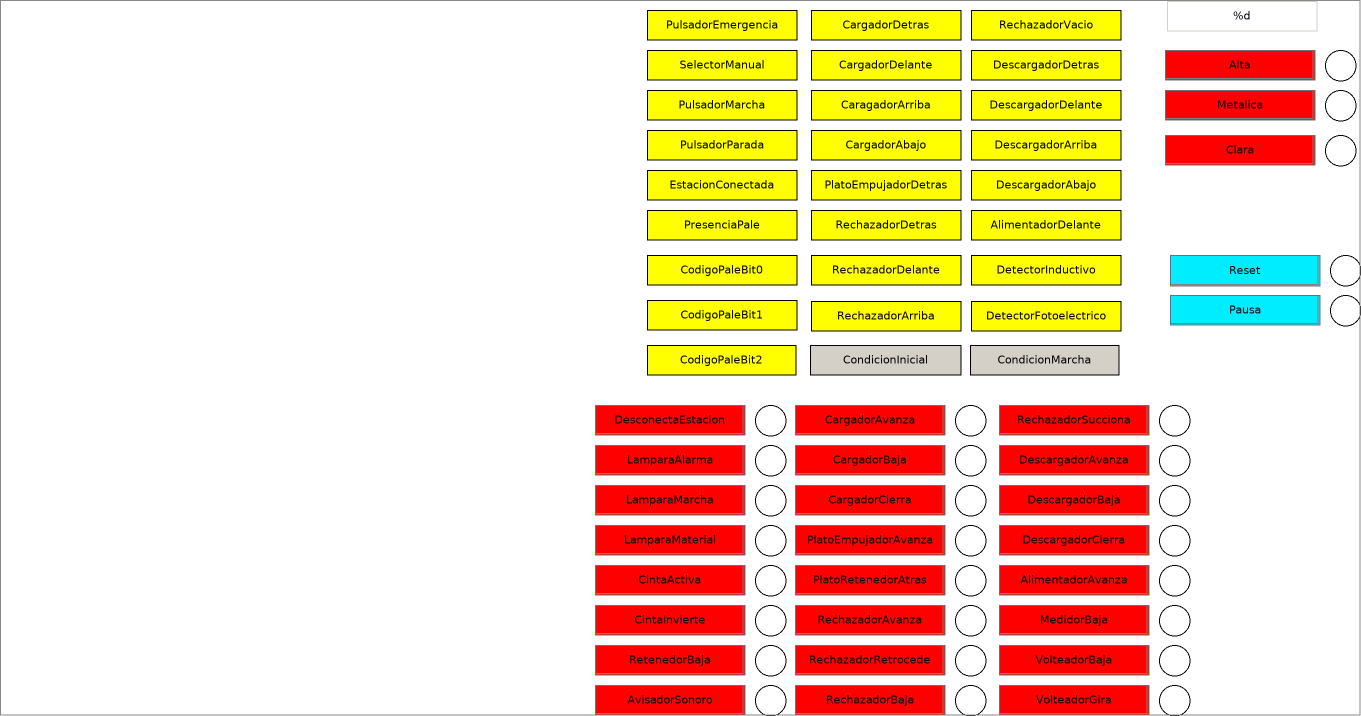
VISUALIZATION Visualization  // 1361x716
    Rectangle (647,170 150x30), "EstacionConectada", colour toggle: MAIN.Estacion.EstacionConectada
        toggle MAIN.Estacion.EstacionConectada
    Rectangle (647,210 150x30), "PresenciaPale", colour toggle: MAIN.Estacion.PresenciaPale
        toggle MAIN.Estacion.PresenciaPale
    Rectangle (647,255 150x30), "CodigoPaleBit0", colour toggle: MAIN.Estacion.CodigoPaleBit0
        toggle MAIN.Estacion.CodigoPaleBit0
    Rectangle (647,300 150x30), "CodigoPaleBit1", colour toggle: MAIN.Estacion.CodigoPaleBit1
        toggle MAIN.Estacion.CodigoPaleBit1
    Rectangle (647,345 149x30), "CodigoPaleBit2", colour toggle: MAIN.Estacion.CodigoPaleBit2
        toggle MAIN.Estacion.CodigoPaleBit2
    Rectangle (647,130 150x30), "PulsadorParada", colour toggle: MAIN.Estacion.PulsadorParada
        toggle MAIN.Estacion.PulsadorParada
    Rectangle (647,90 150x30), "PulsadorMarcha", colour toggle: MAIN.Estacion.PulsadorMarcha
        toggle MAIN.Estacion.PulsadorMarcha
    Rectangle (647,50 150x30), "SelectorManual", colour toggle: MAIN.Estacion.SelectorManual
        toggle MAIN.Estacion.SelectorManual
    Rectangle (647,10 150x30), "PulsadorEmergencia", colour toggle: MAIN.Estacion.PulsadorEmergencia
        toggle MAIN.Estacion.PulsadorEmergencia
    Rectangle (811,170 150x30), "PlatoEmpujadorDetras", colour toggle: MAIN.Estacion.PlatoEmpujadorDetras
        toggle MAIN.Estacion.PlatoEmpujadorDetras
    Rectangle (811,210 150x30), "RechazadorDetras", colour toggle: MAIN.Estacion.RechazadorDetras
        toggle MAIN.Estacion.RechazadorDetras
    Rectangle (811,255 150x30), "RechazadorDelante", colour toggle: MAIN.Estacion.RechazadorDelante
        toggle MAIN.Estacion.RechazadorDelante
    Rectangle (811,130 150x30), "CargadorAbajo", colour toggle: MAIN.Estacion.CargadorAbajo
        toggle MAIN.Estacion.CargadorAbajo
    Rectangle (811,90 150x30), "CaragadorArriba", colour toggle: MAIN.Estacion.CargadorArriba
        toggle MAIN.Estacion.CargadorArriba
    Rectangle (811,50 150x30), "CargadorDelante", colour toggle: MAIN.Estacion.CargadorDelante
        toggle MAIN.Estacion.CargadorDelante
    Rectangle (811,10 150x30), "CargadorDetras", colour toggle: MAIN.Estacion.CargadorDetras
        toggle MAIN.Estacion.CargadorDetras
    Rectangle (811,301 150x30), "RechazadorArriba", colour toggle: MAIN.Estacion.RechazadorArriba
        toggle MAIN.Estacion.RechazadorArriba
    Rectangle (971,170 150x30), "DescargadorAbajo", colour toggle: MAIN.Estacion.DescargadorAbajo
        toggle MAIN.Estacion.DescargadorAbajo
    Rectangle (971,210 150x30), "AlimentadorDelante", colour toggle: MAIN.Estacion.AlimentadorDelante
        toggle MAIN.Estacion.AlimentadorDelante
    Rectangle (971,255 150x30), "DetectorInductivo", colour toggle: MAIN.Estacion.DetectorInductivo
        toggle MAIN.Estacion.DetectorInductivo
    Rectangle (971,130 150x30), "DescargadorArriba", colour toggle: MAIN.Estacion.DescargadorArriba
        toggle MAIN.Estacion.DescargadorArriba
    Rectangle (971,90 150x30), "DescargadorDelante", colour toggle: MAIN.Estacion.DescargadorDelante
        toggle MAIN.Estacion.DescargadorDelante
    Rectangle (971,50 150x30), "DescargadorDetras", colour toggle: MAIN.Estacion.DescargadorDetras
        toggle MAIN.Estacion.DescargadorDetras
    Rectangle (971,10 150x30), "RechazadorVacio", colour toggle: MAIN.Estacion.RechazadorVacio
        toggle MAIN.Estacion.RechazadorVacio
    Rectangle (971,301 150x30), "DetectorFotoelectrico", colour toggle: MAIN.Estacion.DetectorFotoelectrico
        toggle MAIN.Estacion.DetectorFotoelectrico
    Rectangle (810,345 151x30), "CondicionInicial", colour toggle: MAIN.Estacion.CondicionInicial
        toggle MAIN.Estacion.CondicionInicial
    Rectangle (970,345 149x30), "CondicionMarcha", colour toggle: MAIN.Estacion.CondicionMarcha
        toggle MAIN.Estacion.CondicionMarcha
    Button (595,445 150x30), "LamparaAlarma"
        toggle MAIN.Estacion.LamparaAlarma
    Ellipse (755,445 31x31), colour toggle: MAIN.Estacion.LamparaAlarma
    Button (595,405 150x30), "DesconectaEstacion"
        toggle MAIN.Estacion.DesconectaEstacion
    Ellipse (755,405 31x31), colour toggle: MAIN.Estacion.DesconectaEstacion
    Button (595,525 150x30), "LamparaMaterial"
        toggle MAIN.Estacion.LamparaMaterial
    Ellipse (755,525 31x31), colour toggle: MAIN.Estacion.LamparaMaterial
    Button (595,485 150x30), "LamparaMarcha"
        toggle MAIN.Estacion.LamparaMarcha
    Ellipse (755,485 31x31), colour toggle: MAIN.Estacion.LamparaMarcha
    Button (595,605 150x30), "CintaInvierte"
        toggle MAIN.Estacion.CintaInvierte
    Ellipse (755,605 31x31), colour toggle: MAIN.Estacion.CintaInvierte
    Button (595,565 150x30), "CintaActiva"
        toggle MAIN.Estacion.CintaActiva
    Ellipse (755,565 31x31), colour toggle: MAIN.Estacion.CintaActiva
    Button (595,685 150x30), "AvisadorSonoro"
        toggle MAIN.Estacion.AvisadorSonoro
    Ellipse (755,685 31x31), colour toggle: MAIN.Estacion.AvisadorSonoro
    Button (595,645 150x30), "RetenedorBaja"
        toggle MAIN.Estacion.RetenedorBaja
    Ellipse (755,645 31x31), colour toggle: MAIN.Estacion.RetenedorBaja
    Button (795,445 150x30), "CargadorBaja"
        toggle MAIN.Estacion.CargadorBaja
    Ellipse (955,445 31x31), colour toggle: MAIN.Estacion.CargadorBaja
    Button (795,405 150x30), "CargadorAvanza"
        toggle MAIN.Estacion.CargadorAvanza
    Ellipse (955,405 31x31), colour toggle: MAIN.Estacion.CargadorAvanza
    Button (795,525 150x30), "PlatoEmpujadorAvanza"
        toggle MAIN.Estacion.PlatoEmpujadorAvanza
    Ellipse (955,525 31x31), colour toggle: MAIN.Estacion.PlatoEmpujadorAvanza
    Button (795,485 150x30), "CargadorCierra"
        toggle MAIN.Estacion.CargadorCierra
    Ellipse (955,485 31x31), colour toggle: MAIN.Estacion.CargadorCierra
    Button (795,605 150x30), "RechazadorAvanza"
        toggle MAIN.Estacion.RechazadorAvanza
    Ellipse (955,605 31x31), colour toggle: MAIN.Estacion.RechazadorAvanza
    Button (795,565 150x30), "PlatoRetenedorAtras"
        toggle MAIN.Estacion.PlatoRetenedorAtras
    Ellipse (955,565 31x31), colour toggle: MAIN.Estacion.PlatoRetenedorAtras
    Button (795,685 150x30), "RechazadorBaja"
        toggle MAIN.Estacion.RechazadorBaja
    Ellipse (955,685 31x31), colour toggle: MAIN.Estacion.RechazadorBaja
    Button (795,645 150x30), "RechazadorRetrocede"
        toggle MAIN.Estacion.RechazadorRetrocede
    Ellipse (955,645 31x31), colour toggle: MAIN.Estacion.RechazadorRetrocede
    Button (999,445 150x30), "DescargadorAvanza"
        toggle MAIN.Estacion.DescargadorAvanza
    Ellipse (1159,445 31x31), colour toggle: MAIN.Estacion.DescargadorAvanza
    Button (999,405 150x30), "RechazadorSucciona"
        toggle MAIN.Estacion.RechazadorSucciona
    Ellipse (1159,405 31x31), colour toggle: MAIN.Estacion.RechazadorSucciona
    Button (999,525 150x30), "DescargadorCierra"
        toggle MAIN.Estacion.DescargadorCierra
    Ellipse (1159,525 31x31), colour toggle: MAIN.Estacion.DescargadorCierra
    Button (999,485 150x30), "DescargadorBaja"
        toggle MAIN.Estacion.DescargadorBaja
    Ellipse (1159,485 31x31), colour toggle: MAIN.Estacion.DescargadorBaja
    Button (999,605 150x30), "MedidorBaja"
        toggle MAIN.Estacion.MedidorBaja
    Ellipse (1159,605 31x31), colour toggle: MAIN.Estacion.MedidorBaja
    Button (999,565 150x30), "AlimentadorAvanza"
        toggle MAIN.Estacion.AlimentadorAvanza
    Ellipse (1159,565 31x31), colour toggle: MAIN.Estacion.AlimentadorAvanza
    Button (999,685 150x30), "VolteadorGira"
        toggle MAIN.Estacion.VolteadorGira
    Ellipse (1159,685 31x31), colour toggle: MAIN.Estacion.VolteadorGira
    Button (999,645 150x30), "VolteadorBaja"
        toggle MAIN.Estacion.VolteadorBaja
    Ellipse (1159,645 31x31), colour toggle: MAIN.Estacion.VolteadorBaja
    Button (1165,50 150x30), "Alta"
        toggle MAIN.Estacion.TapaDeseada.Alta
    Ellipse (1325,50 31x31), colour toggle: MAIN.Estacion.TapaDeseada.Alta
    Button (1165,90 150x30), "Metalica"
        toggle MAIN.Estacion.TapaDeseada.Metalica
    Ellipse (1325,90 31x31), colour toggle: MAIN.Estacion.TapaDeseada.Metalica
    Button (1165,135 150x30), "Clara"
        toggle MAIN.Estacion.TapaDeseada.Clara
    Ellipse (1325,135 31x31), colour toggle: MAIN.Estacion.TapaDeseada.Clara
    Textfield (1167,1 150x30), "%d", text variable: MAIN.Estacion.NumPiezasDes
        OnMouseClick: write the text variable via Default
    Button (1170,295 150x30), "Pausa"
        toggle MAIN.Estacion.PausaEstado
    Ellipse (1330,295 31x31), colour toggle: MAIN.Estacion.PausaEstado
    Button (1170,255 150x31), "Reset"
        toggle MAIN.Estacion.ReiniciaEstado
    Ellipse (1330,255 31x31), colour toggle: MAIN.Estacion.ReiniciaEstado
END_VISUALIZATION

(* stored: Version 1.1.0.1, ProductVersion 3.1.4024.12
   Visu Visualization: Id {d673722a-6320-49a9-8529-10ae53f6d6d1} *)
